Yaskawa INFORM job: X2_24A(90,180).JBI

/JOB
//NAME X2_24A(90,180)
///FOLDERNAME X2
//POS
///NPOS 99,99,99,6,0,0
///TOOL 0
///POSTYPE PULSE
///PULSE
C00000=-2000,-92772,-84335,0,66375,0
C00001=61786,-92772,-84335,2347,66375,-79401
C00002=102277,-27188,-81237,-24448,94316,-80884
C00003=97244,21725,-41177,-22449,93615,-82233
C00004=95530,462,4396,-55956,36816,-51794
C00005=94424,6187,12285,-57576,35067,-50925
C00006=93996,8571,15581,-58338,34366,-50524
C00007=93996,9261,17575,-59445,33898,-49925
C00008=93996,8571,15581,-58338,34366,-50524
C00009=93267,12817,19373,-58151,33839,-50654
C00010=93996,8571,15581,-58338,34366,-50524
C00011=95521,1087,6495,-57044,36258,-51187
C00012=96592,2869,6453,-65825,56052,-48227
C00013=94772,6998,13020,-66731,54034,-47573
C00014=94060,8748,15768,-67150,53233,-47286
C00015=94060,9552,18085,-67847,52819,-46755
C00016=94060,8748,15768,-67150,53233,-47286
C00017=92626,10057,16930,-66950,52266,-47512
C00018=94060,8748,15768,-67150,53233,-47286
C00019=96573,3490,8496,-66397,55638,-47762
C00020=83582,5061,8367,-59913,58634,-65118
C00021=81471,7687,13629,-60535,56339,-64672
C00022=80635,8836,15839,-60828,55424,-64478
C00023=80635,9690,18292,-61474,54884,-63961
C00024=80635,8836,15839,-60828,55424,-64478
C00025=79828,9033,16014,-60679,54915,-64642
C00026=80635,8836,15839,-60828,55424,-64478
C00027=83597,5664,10366,-60398,58167,-64691
C00028=83314,10150,12730,-59594,89568,-59936
C00029=81399,9267,14976,-59682,87415,-59552
C00030=81014,9626,17081,-59725,86592,-59179
C00031=81014,10332,19089,-59751,86136,-58834
C00032=81014,9626,17081,-59725,86592,-59179
C00033=80226,8223,15841,-59775,86122,-59334
C00034=81014,9626,17081,-59725,86592,-59179
C00035=83301,10774,14815,-59578,89053,-59559
C00036=98806,-6617,-7331,-59053,101140,-58606
C00037=97102,-16285,-8510,-58460,97807,-57230
C00038=95610,-19203,-5710,-58231,95144,-56240
C00039=95610,-18645,-4180,-58161,94786,-55981
C00040=96019,-16166,-2121,-59216,96428,-56839
C00041=95765,-17656,-3227,-59244,96227,-56851
C00042=96019,-16166,-2121,-59216,96428,-56839
C00043=98806,-6617,-7331,-59053,101140,-58606
C00044=83650,45812,10891,-63097,77396,-50083
C00045=82040,46827,21520,-63951,73569,-47805
C00046=81304,48087,22594,-63748,73022,-47936
C00047=82382,46154,21930,-64152,73438,-47516
C00048=81304,48079,23723,-63930,72698,-47640
C00049=81325,48203,23856,-63940,72703,-47628
C00050=80528,45970,21634,-59995,63959,-50181
C00051=80159,45513,21016,-56886,58795,-52013
C00052=79561,44924,20521,-53542,54142,-53866
C00053=80930,50792,26842,-52633,51858,-54251
C00054=80922,51336,27332,-50501,49586,-55378
C00055=80906,51749,27861,-49613,48546,-55836
C00056=80960,51889,27980,-48874,47816,-56226
C00057=80899,52077,28242,-47421,46344,-56985
C00058=81070,52679,28952,-47614,46346,-56872
C00059=80548,47424,22156,-44596,45760,-58565
C00060=81458,42877,14387,-43611,47989,-59314
C00061=91002,51772,6505,-49273,82170,-67204
C00062=101987,13091,-892,-55645,108662,-64355
C00063=110253,6769,-1127,-53677,111646,-61313
C00064=109069,2020,-4496,-53719,110740,-61430
C00065=109385,7501,2227,-53217,110114,-60832
C00066=109192,2312,-2241,-53275,110054,-60910
C00067=100675,7131,2033,-54353,105017,-62710
C00068=100597,7181,2077,-54362,104971,-62725
C00069=98280,5172,14,-55265,98555,-65123
C00070=92725,-3156,-6815,-54418,80144,-71316
C00071=87235,-4368,-7735,-50596,66698,-76420
C00072=92539,-2221,-10635,-51205,72117,-76021
C00073=96871,14274,1468,-54076,82371,-72764
C00074=94701,9031,3178,-59274,52046,-46005
C00075=93342,13775,10378,-60199,50156,-45313
C00076=92447,15859,11447,-59599,49816,-45723
C00077=93434,13866,11409,-60652,49914,-44989
C00078=92673,17069,14252,-60484,49385,-45106
C00079=92707,17100,14281,-60496,49406,-45098
C00080=95769,24674,21440,-57601,43614,-47021
C00081=97283,25037,21490,-42917,31085,-55304
C00082=96416,20010,16135,-41713,31228,-55971
C00083=96977,14076,7690,-40003,33138,-56882
C00084=85021,42815,2038,-36976,67324,-74168
C00085=87037,99,-8557,-56339,77378,-69862
C00086=84861,88,-5624,-56340,75042,-69589
C00087=84770,-1894,-7034,-56357,74898,-69547
C00088=86315,-1244,-5605,-56691,75514,-69027
C00089=84898,-1236,-5744,-56471,74715,-69344
C00090=84911,-1174,-5693,-56473,74723,-69341
C00091=83726,13860,7501,-56385,73791,-69419
C00092=81991,21696,14871,-53905,65164,-72191
C00093=78866,22111,15159,-45765,51452,-78645
C00094=78646,18844,10981,-44406,51004,-79638
C00095=80451,15982,5388,-44195,53341,-79866
C00096=99337,20331,-42513,-23301,94176,-81727
C00097=89347,-122219,-94568,-8337,58557,-68745
C00098=-2000,-92772,-84335,0,66375,0
BC00000=244938,523905,804554
BC00001=244938,517847,286212
BC00002=244938,493983,17
BC00003=244938,493983,17
BC00004=305514,414637,205828
BC00005=305514,414637,205828
BC00006=305514,414637,205828
BC00007=305514,414637,205828
BC00008=305514,414637,205828
BC00009=305514,414637,205828
BC00010=305514,414637,205828
BC00011=305514,414637,205828
BC00012=306843,429968,205896
BC00013=306843,429968,205896
BC00014=306843,429968,205896
BC00015=306843,429968,205896
BC00016=306843,429968,205896
BC00017=306843,429968,205896
BC00018=306843,429968,205896
BC00019=306843,429968,205896
BC00020=266221,447545,232190
BC00021=266221,447545,232190
BC00022=266221,447545,232190
BC00023=266221,447545,232190
BC00024=266221,447545,232190
BC00025=266221,447545,232190
BC00026=266221,447545,232190
BC00027=266221,447545,232190
BC00028=250481,433829,248791
BC00029=250481,433829,248791
BC00030=250481,433829,248791
BC00031=250481,433829,248791
BC00032=250481,433829,248791
BC00033=250481,433829,248791
BC00034=250481,433829,248791
BC00035=250481,433829,248791
BC00036=250481,433829,248791
BC00037=250481,433829,248791
BC00038=250481,433829,248791
BC00039=250481,433829,248791
BC00040=250481,433829,248791
BC00041=250481,433829,248791
BC00042=250481,433829,248791
BC00043=250481,433829,248791
BC00044=252129,446239,17
BC00045=252129,446239,17
BC00046=252129,446239,17
BC00047=252129,446239,17
BC00048=252129,446239,16
BC00049=252129,446239,16
BC00050=252129,446239,17
BC00051=252129,446239,17
BC00052=252129,446239,17
BC00053=252129,446239,17
BC00054=252129,446239,17
BC00055=252129,446239,17
BC00056=252129,446239,17
BC00057=252129,446239,17
BC00058=252129,446239,17
BC00059=252129,446239,17
BC00060=252129,446239,17
BC00061=254149,484604,17
BC00062=278420,467745,176006
BC00063=278420,467745,176006
BC00064=278420,467745,176006
BC00065=278420,467745,176006
BC00066=278420,467745,176006
BC00067=278420,467745,176006
BC00068=278420,467745,176006
BC00069=278420,467745,176006
BC00070=278420,467745,176004
BC00071=278420,467745,176006
BC00072=278420,467745,176006
BC00073=278420,467745,176006
BC00074=300781,423407,142570
BC00075=300781,423407,142570
BC00076=300781,423407,142564
BC00077=300781,423407,142564
BC00078=300781,423407,142564
BC00079=300781,423407,142564
BC00080=300781,423407,142570
BC00081=300781,423407,142570
BC00082=300781,423407,142570
BC00083=300781,423407,142570
BC00084=248642,475261,17
BC00085=269856,449889,162337
BC00086=269856,449889,162337
BC00087=269856,449889,162337
BC00088=269856,449889,162337
BC00089=269856,449889,162337
BC00090=269856,449889,162337
BC00091=269856,449889,162337
BC00092=269856,449889,162337
BC00093=269856,449889,162337
BC00094=269856,449889,162337
BC00095=269856,449889,162337
BC00096=244938,493983,17
BC00097=244938,517847,286212
BC00098=244938,523905,804554
EC00000=-798156,-1296783
EC00001=-798156,-1296783
EC00002=-798156,-1296783
EC00003=-798156,-1296783
EC00004=-798156,-1296783
EC00005=-798156,-1296783
EC00006=-798156,-1296783
EC00007=-798156,-1296783
EC00008=-798156,-1296783
EC00009=-798156,-1296783
EC00010=-798156,-1296783
EC00011=-798156,-1296783
EC00012=-798156,-1296783
EC00013=-798156,-1296783
EC00014=-798156,-1296783
EC00015=-798156,-1296783
EC00016=-798156,-1296783
EC00017=-798156,-1296783
EC00018=-798156,-1296783
EC00019=-798156,-1296783
EC00020=-798156,-1296783
EC00021=-798156,-1296783
EC00022=-798156,-1296783
EC00023=-798156,-1296783
EC00024=-798156,-1296783
EC00025=-798156,-1296783
EC00026=-798156,-1296783
EC00027=-798156,-1296783
EC00028=-798156,-1296783
EC00029=-798156,-1296783
EC00030=-798156,-1296783
EC00031=-798156,-1296783
EC00032=-798156,-1296783
EC00033=-798156,-1296783
EC00034=-798156,-1296783
EC00035=-798156,-1296783
EC00036=-798156,-1296783
EC00037=-798156,-1296783
EC00038=-798156,-1296783
EC00039=-798156,-1296783
EC00040=-798156,-1296783
EC00041=-798156,-1296783
EC00042=-798156,-1296783
EC00043=-798156,-1296783
EC00044=-798156,-1296783
EC00045=-798156,-1296783
EC00046=-798156,-1296783
EC00047=-798156,-1296783
EC00048=-798155,-1296782
EC00049=-798155,-1296782
EC00050=-798156,-1296783
EC00051=-798156,-1296783
EC00052=-798156,-1296783
EC00053=-798156,-1296783
EC00054=-798156,-1296783
EC00055=-798156,-1296783
EC00056=-798156,-1296783
EC00057=-798156,-1296783
EC00058=-798156,-1296783
EC00059=-798156,-1296783
EC00060=-798156,-1296783
EC00061=-798156,-1296783
EC00062=-798156,-1296783
EC00063=-798156,-1296783
EC00064=-798156,-1296783
EC00065=-798156,-1296783
EC00066=-798156,-1296783
EC00067=-798156,-1296783
EC00068=-798156,-1296783
EC00069=-798156,-1296783
EC00070=-798155,-1296782
EC00071=-798156,-1296783
EC00072=-798156,-1296783
EC00073=-798156,-1296783
EC00074=-798156,-1296783
EC00075=-798156,-1296783
EC00076=-798154,-1296781
EC00077=-798154,-1296781
EC00078=-798154,-1296781
EC00079=-798154,-1296781
EC00080=-798156,-1296783
EC00081=-798156,-1296783
EC00082=-798156,-1296783
EC00083=-798156,-1296783
EC00084=-798156,-1296783
EC00085=-798156,-1296783
EC00086=-798156,-1296783
EC00087=-798156,-1296783
EC00088=-798156,-1296783
EC00089=-798156,-1296783
EC00090=-798156,-1296783
EC00091=-798156,-1296783
EC00092=-798156,-1296783
EC00093=-798156,-1296783
EC00094=-798156,-1296783
EC00095=-798156,-1296783
EC00096=-798156,-1296783
EC00097=-798156,-1296783
EC00098=-798156,-1296783
///POSTYPE BASE
///RECTAN
///RCONF 0,0,0,0,1,0,0,0,0,0,0,0,0,0,0,0,0,0,0,0,0,0,0,0
P00006=2.006,1.622,-0.565,0.0000,0.0000,0.0000
P00021=0.073,2.058,-0.109,0.0000,0.0000,0.0000
P00022=2.006,1.622,-0.565,0.0000,0.0000,0.0000
///RCONF 0,0,0,0,0,0,0,0,0,0,0,0,0,0,0,0,0,0,0,0,0,0,0,0
P00023=-2.957,-4.083,2.762,0.0000,0.0000,0.0000
P00024=-1.466,-0.226,-0.419,0.0000,0.0000,0.0000
P00025=3.643,0.007,-2.585,0.0000,0.0000,0.0000
//INST
///DATE 2024/12/03 13:27
///ATTR SC,RW
///GROUP1 RB1,BS1
///GROUP2 ST1
NOP
'X2_24A(90,180)
MOVJ C00000 BC00000 VJ=100.00  +MOVJ EC00000 VJ=100.00
MOVJ C00001 BC00001 VJ=100.00  +MOVJ EC00001 VJ=100.00
MOVJ C00002 BC00002 VJ=100.00  +MOVJ EC00002 VJ=100.00
MOVJ C00003 BC00003 VJ=100.00  +MOVJ EC00003 VJ=100.00
'Path S3533
SFTOF3D
MOVJ C00004 BC00004 VJ=100.00  +MOVJ EC00004 VJ=100.00
MOVL C00005 BC00005 V=800.0  +MOVJ EC00005 VJ=100.00
SMOVL C00006 BC00006 V=166.7  +MOVJ EC00006
SREFP 3 C00007 BC00007  +REFP EC00007
CALL JOB:SEARCH-R1-S13D
SET P021 P006
SFTON3D P021
SMOVL C00008 BC00008 V=166.7  +MOVJ EC00008
SREFP 3 C00009 BC00009  +REFP EC00009
CALL JOB:SEARCH-R1-S13D
SET P021 P006
SFTON3D P021
SMOVL C00010 BC00010 V=166.7  +MOVJ EC00010
MOVL C00011 BC00011 V=1000.0  +MOVJ EC00011 VJ=100.00
'EndPath S3533
'Path S3534
SFTOF3D
MOVJ C00012 BC00012 VJ=100.00  +MOVJ EC00012 VJ=100.00
MOVL C00013 BC00013 V=800.0  +MOVJ EC00013 VJ=100.00
SMOVL C00014 BC00014 V=166.7  +MOVJ EC00014
SREFP 3 C00015 BC00015  +REFP EC00015
CALL JOB:SEARCH-R1-S13D
SET P022 P006
SFTON3D P022
SMOVL C00016 BC00016 V=166.7  +MOVJ EC00016
SREFP 3 C00017 BC00017  +REFP EC00017
CALL JOB:SEARCH-R1-S13D
SET P022 P006
SFTON3D P022
SMOVL C00018 BC00018 V=166.7  +MOVJ EC00018
MOVL C00019 BC00019 V=1000.0  +MOVJ EC00019 VJ=100.00
'EndPath S3534
'Path S3535
SFTOF3D
MOVJ C00020 BC00020 VJ=100.00  +MOVJ EC00020 VJ=100.00
MOVL C00021 BC00021 V=800.0  +MOVJ EC00021 VJ=100.00
SMOVL C00022 BC00022 V=166.7  +MOVJ EC00022
SREFP 3 C00023 BC00023  +REFP EC00023
CALL JOB:SEARCH-R1-S13D
SET P023 P006
SFTON3D P023
SMOVL C00024 BC00024 V=166.7  +MOVJ EC00024
SREFP 3 C00025 BC00025  +REFP EC00025
CALL JOB:SEARCH-R1-S13D
SET P023 P006
SFTON3D P023
SMOVL C00026 BC00026 V=166.7  +MOVJ EC00026
MOVL C00027 BC00027 V=1000.0  +MOVJ EC00027 VJ=100.00
'EndPath S3535
'Path S3536
SFTOF3D
MOVJ C00028 BC00028 VJ=100.00  +MOVJ EC00028 VJ=100.00
MOVL C00029 BC00029 V=800.0  +MOVJ EC00029 VJ=100.00
SMOVL C00030 BC00030 V=166.7  +MOVJ EC00030
SREFP 3 C00031 BC00031  +REFP EC00031
CALL JOB:SEARCH-R1-S13D
SET P024 P006
SFTON3D P024
SMOVL C00032 BC00032 V=166.7  +MOVJ EC00032
SREFP 3 C00033 BC00033  +REFP EC00033
CALL JOB:SEARCH-R1-S13D
SET P024 P006
SFTON3D P024
SMOVL C00034 BC00034 V=166.7  +MOVJ EC00034
MOVL C00035 BC00035 V=1000.0  +MOVJ EC00035 VJ=100.00
'EndPath S3536
'Path W3537
SFTOF3D
MOVJ C00036 BC00036 VJ=100.00  +MOVJ EC00036 VJ=100.00
MOVL C00037 BC00037 V=800.0  +MOVJ EC00037 VJ=100.00
SMOVL C00038 BC00038 V=166.7  +MOVJ EC00038
SREFP 3 C00039 BC00039  +REFP EC00039
CALL JOB:SEARCH-R1-S13D
SET P025 P006
SFTON3D P025
SMOVL C00040 BC00040 V=166.7  +MOVJ EC00040
SREFP 3 C00041 BC00041  +REFP EC00041
CALL JOB:SEARCH-R1-S13D
SET P025 P006
SFTON3D P025
SMOVL C00042 BC00042 V=166.7  +MOVJ EC00042
MOVL C00043 BC00043 V=1000.0  +MOVJ EC00043 VJ=100.00
SFTOF3D
SFTON3D P022
MOVJ C00044 BC00044 VJ=100.00  +MOVJ EC00044 VJ=100.00
SMOVL C00045 BC00045 V=800.0  +MOVJ EC00045
SREFP 1 C00046 BC00046  +REFP EC00046
SREFP 2 C00047 BC00047  +REFP EC00047
SMOVL C00048 BC00048 V=150.0 PL=0  +MOVJ EC00048
MACRO1 MJ#(0) ARGF21
ARCON
SWVON WEV#(100)
SMOVC C00049 BC00049 V=9.2  +MOVJ EC00049
SMOVC C00050 BC00050 V=9.2  +MOVJ EC00050
SMOVC C00051 BC00051 V=9.2  +MOVJ EC00051
SMOVC C00052 BC00052 V=9.2  +MOVJ EC00052
SMOVC C00053 BC00053 V=9.2  +MOVJ EC00053
ARCON
SWVON WEV#(100)
SMOVC C00054 BC00054 V=9.2  +MOVJ EC00054
SMOVC C00055 BC00055 V=9.2  +MOVJ EC00055
SMOVC C00056 BC00056 V=9.2  +MOVJ EC00056
SMOVC C00057 BC00057 V=9.2  +MOVJ EC00057
SMOVC C00058 BC00058 V=9.2  +MOVJ EC00058
ARCOF
SWVOF
SMOVL C00059 BC00059 V=800.0  +MOVJ EC00059
SMOVL C00060 BC00060 V=1000.0  +MOVJ EC00060
SFTOF3D
'EndPath W3537
MOVJ C00061 BC00061 VJ=100.00  +MOVJ EC00061 VJ=100.00
'Path W3538
SFTOF3D
SFTON3D P025
MOVJ C00062 BC00062 VJ=100.00  +MOVJ EC00062 VJ=100.00
SMOVL C00063 BC00063 V=800.0  +MOVJ EC00063
SREFP 1 C00064 BC00064  +REFP EC00064
SREFP 2 C00065 BC00065  +REFP EC00065
SMOVL C00066 BC00066 V=150.0 PL=0  +MOVJ EC00066
ARCON
SWVON WEV#(100)
SMOVL C00067 BC00067 V=9.2  +MOVJ EC00067
SMOVC C00068 BC00068 V=9.2  +MOVJ EC00068
SFTON3D P024
SMOVC C00069 BC00069 V=9.2  +MOVJ EC00069
SMOVC C00070 BC00070 V=9.2  +MOVJ EC00070
SMOVC C00071 BC00071 V=9.2  +MOVJ EC00071
ARCOF
SWVOF
SMOVL C00072 BC00072 V=800.0  +MOVJ EC00072
SMOVL C00073 BC00073 V=1000.0  +MOVJ EC00073
SFTOF3D
'EndPath W3538
'Path W3539
SFTOF3D
SFTON3D P021
MOVJ C00074 BC00074 VJ=100.00  +MOVJ EC00074 VJ=100.00
SMOVL C00075 BC00075 V=800.0  +MOVJ EC00075
SREFP 1 C00076 BC00076  +REFP EC00076
SREFP 2 C00077 BC00077  +REFP EC00077
SMOVL C00078 BC00078 V=150.0 PL=0  +MOVJ EC00078
ARCON
SWVON WEV#(100)
SMOVC C00079 BC00079 V=9.2  +MOVJ EC00079
SMOVC C00080 BC00080 V=9.2  +MOVJ EC00080
SMOVC C00081 BC00081 V=9.2  +MOVJ EC00081
ARCOF
SWVOF
SMOVL C00082 BC00082 V=800.0  +MOVJ EC00082
SMOVL C00083 BC00083 V=1000.0  +MOVJ EC00083
SFTOF3D
'EndPath W3539
MOVJ C00084 BC00084 VJ=100.00  +MOVJ EC00084 VJ=100.00
'Path W3540
SFTOF3D
SFTON3D P023
MOVJ C00085 BC00085 VJ=100.00  +MOVJ EC00085 VJ=100.00
SMOVL C00086 BC00086 V=800.0  +MOVJ EC00086
SREFP 1 C00087 BC00087  +REFP EC00087
SREFP 2 C00088 BC00088  +REFP EC00088
SMOVL C00089 BC00089 V=166.7 PL=0  +MOVJ EC00089
ARCON
SWVON WEV#(100)
SMOVC C00090 BC00090 V=9.2  +MOVJ EC00090
SMOVC C00091 BC00091 V=9.2  +MOVJ EC00091
SMOVC C00092 BC00092 V=9.2  +MOVJ EC00092
SMOVC C00093 BC00093 V=9.2  +MOVJ EC00093
ARCOF
SWVOF
SMOVL C00094 BC00094 V=800.0  +MOVJ EC00094
SMOVL C00095 BC00095 V=1000.0  +MOVJ EC00095
SFTOF3D
'EndPath W3540
MOVJ C00096 BC00096 VJ=100.00  +MOVJ EC00096 VJ=100.00
MOVJ C00097 BC00097 VJ=100.00  +MOVJ EC00097 VJ=100.00
MOVJ C00098 BC00098 VJ=100.00  +MOVJ EC00098 VJ=100.00
END
